// TIA Portal project "MODBUS" (V17)

(* hardware
DEVICE "S7-1500/ET200MP station_1"  S7-1500 station
   slot 0: "Rail_0"  Rack  6ES7 590-1***0-0AA0
   slot 1: "PLC_1"  CPU 1512C-1 PN  6ES7 512-1CK00-0AB0  V2.1
      slot 3: "CPU display_1"  6ES7591-1AA00-0AA0
      slot 32768: "PROFINET interface_1"  X1
         slot 32769: "Port_1"  X1 P1
         slot 32770: "Port_2"  X1 P2
*)

// ===== PLC "PLC_1"  CPU 1512C-1 PN =====

VAR_GLOBAL   // PLC tag table "Default tag table"
   "System_Byte" AT %MB1 : Byte;
   "FirstScan" AT %M1.0 : Bool;
   "DiagStatusUpdate" AT %M1.1 : Bool;
   "AlwaysTRUE" AT %M1.2 : Bool;
   "AlwaysFALSE" AT %M1.3 : Bool;
   "Clock_Byte" AT %MB0 : Byte;
   "Clock_10Hz" AT %M0.0 : Bool;
   "Clock_5Hz" AT %M0.1 : Bool;
   "Clock_2.5Hz" AT %M0.2 : Bool;
   "Clock_2Hz" AT %M0.3 : Bool;
   "Clock_1.25Hz" AT %M0.4 : Bool;
   "Clock_1Hz" AT %M0.5 : Bool;
   "Clock_0.625Hz" AT %M0.6 : Bool;
   "Clock_0.5Hz" AT %M0.7 : Bool;
END_VAR

DATA_BLOCK "MODBUS-DATA"   // DB9
{ S7_Optimized_Access := 'FALSE' }
VERSION : 0.1
   VAR
      DATA_1_INT : Array[0..10] of Int;
      DATA_2_REAL : Array[0..10] of Real;
   END_VAR
BEGIN
END_DATA_BLOCK

DATA_BLOCK "MODBUS-CLIENT-PARAMETERS"   // DB11
{ S7_Optimized_Access := 'FALSE' }
VERSION : 0.1
   VAR
      CONNECT : TCON_IP_v4;
      REQ : Bool;
      MB_MODE : USInt;
      MB_DATA_ADDR : UDInt := 40001;
      MB_DATA_LEN : UInt := 11;
      DONE : Bool;
      BUSY : Bool;
      ERROR : Bool;
      STATUS : Word;
   END_VAR
BEGIN
   CONNECT.InterfaceId := 64;
   CONNECT.ID := 4;
   CONNECT.ActiveEstablished := true;
   CONNECT.RemoteAddress.ADDR[1] := 192;
   CONNECT.RemoteAddress.ADDR[2] := 168;
   CONNECT.RemoteAddress.ADDR[3] := 2;
   CONNECT.RemoteAddress.ADDR[4] := 177;
   CONNECT.RemotePort := 502;
   CONNECT.ConnectionType := 11;
END_DATA_BLOCK

ORGANIZATION_BLOCK "MODBUS"   // OB1, LAD, ProgramCycle
TITLE = "Main Program Sweep (Cycle)"
{ S7_Optimized_Access := 'TRUE' }
VERSION : 0.1
   VAR_INPUT
      Initial_Call : Bool;   // Initial call of this OB
      Remanence : Bool;   // =True, if remanent data are available
   END_VAR
BEGIN

REGION Network 1: MODBUS FOR CLIENT
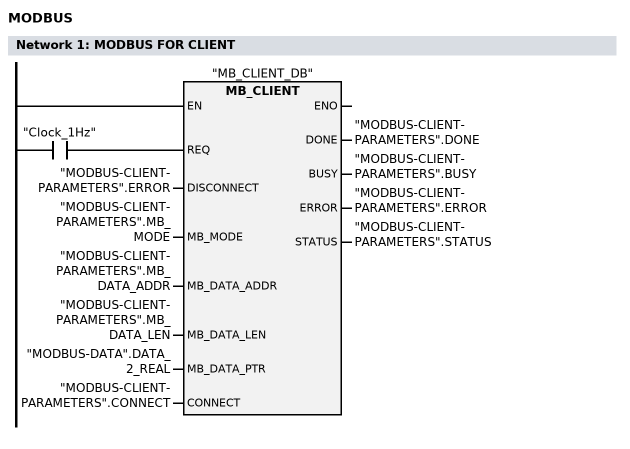
   "MB_CLIENT_DB"(REQ := "Clock_1Hz",   // MB_CLIENT
                  DISCONNECT := "MODBUS-CLIENT-PARAMETERS".ERROR,
                  MB_MODE := "MODBUS-CLIENT-PARAMETERS".MB_MODE,
                  MB_DATA_ADDR := "MODBUS-CLIENT-PARAMETERS".MB_DATA_ADDR,
                  MB_DATA_LEN := "MODBUS-CLIENT-PARAMETERS".MB_DATA_LEN,
                  MB_DATA_PTR := "MODBUS-DATA".DATA_2_REAL,
                  CONNECT := "MODBUS-CLIENT-PARAMETERS".CONNECT,
                  DONE => "MODBUS-CLIENT-PARAMETERS".DONE,
                  BUSY => "MODBUS-CLIENT-PARAMETERS".BUSY,
                  ERROR => "MODBUS-CLIENT-PARAMETERS".ERROR,
                  STATUS => "MODBUS-CLIENT-PARAMETERS".STATUS);
END_REGION
END_ORGANIZATION_BLOCK